PROGRAM P_1Start
VAR
	nState: INT;
	
END_VAR

VAR CONSTANT
	//Here we define our constant where we want the different positon to be. This is instead of making steps you can call this fixed steps.
	Standby    : INT := 00;
	Start		:INT := 01;
	atEntry    : INT := 10;
	Moving     : INT := 20;
	MovingStop : INT := 22;
	Waiting    : INT := 30;
	Stopping   : INT := 40;
	Resetting  : INT := 50;
	Estop      : INT := 99;
		
END_VAR

// This is our first program in the program we have made a state mashine  ( Case ... of ) to define what our system should do
// in the different states.



CASE nState OF
	Standby:		
		IF FIO.bEbStart=TRUE THEN
			FIO.bInEmitBase:=TRUE;
			nState:=Start;
		END_IF
		
	Start: // This is where we declair what should happen if a operator have turned the mashine in auto and pressed start.
			FIO.bInEmitBlueLid:=FALSE;
			FIO.bInEmitGreenLid:=FALSE;
			FIO.bInEmitMetalLid:=FALSE;
			
			
		IF FIO.bEbStart=TRUE AND FIO.bEbAuto=TRUE THEN 
			FIO.bInEmitBlueLid:=TRUE;     //Lids will start to spawn 
			FIO.bInEmitGreenLid:=TRUE;
			FIO.bInEmitMetalLid:=TRUE;
			nState:=Moving;
		END_IF

	Moving:	 //when the lids 
		IF FIO.bInEmitBlueLid=TRUE AND FIO.bInPaSensBlue=FALSE THEN
			FIO.bInConvBlue:=TRUE;       
		END_IF
		IF	FIO.bInEmitGreenLid=TRUE AND FIO.bInPaSensGreen=FALSE THEN
			FIO.bInConvGreen:=TRUE;
		END_IF
		IF FIO.bInEmitMetalLid=TRUE AND FIO.bInPaSensMetal=FALSE THEN
			FIO.bInConvMetal:=TRUE;
		END_IF	
			nState:=MovingStop;
			
	MovingStop:		
	 	IF FIO.bInPaSensBlue=TRUE THEN  
			FIO.bInConvBlue:=FALSE;
		END_IF
		IF FIO.bInPaSensGreen=TRUE THEN	
			FIO.bInConvGreen:=FALSE;
		END_IF	
		IF FIO.bInPaSensMetal=TRUE THEN	
			FIO.bInConvMetal:=FALSE;
		END_IF		
			nState := Waiting;			

		
//----------------------------------------------------------------------------//
	Waiting:
			nState:=Moving;
		
//----------------------------------------------------------------------------//
	Stopping:   //when stop is pressed we move into this statement the stop light turn on / This is also the state we start in when we turn on the PLC /System
		IF FIO.bEbStop = FALSE THEN
			FIO.bEbStopLight:=TRUE;
			FIO.bInEmitBase:=FALSE;
		ELSIF FIO.bEbReset=TRUE THEN
			FIO.bEbStopLight:=FALSE;
			nState:=Standby;	
		END_IF
//----------------------------------------------------------------------------//
			
			
		
//----------------------------------------------------------------------------// 			
	ELSE
			nState:=9999;				
END_CASE

IF NOT FIO.bEbStop THEN  
		nState:=Stopping;	
END_IF

END_PROGRAM

(* stored: Version 1.1.0.1, ProductVersion 3.1.4024.3
   POU P_1Start: Id {fc2519c9-1115-49a1-8835-254105b865d4}, SpecialFunc None *)
